Fanuc KAREL source: kt00993.KL

-- PROVISIONAL review KL for V770-1; original PC SHA256 12c16eac051c8f9e1ecef42b03a925e4016cb3948922b7bc4d866e11e08eff63
-- Incomplete behavior may be omitted. Consult companion uncertainty JSON. Do not deploy.
PROGRAM KT00993
%NOLOCKGROUP
VAR
  X : REAL
  Y : REAL
  Z : REAL
  W : REAL
  P : REAL
  R : REAL
-- UNRESOLVED_DECL P1 type=000106
-- UNRESOLVED_DECL P2 type=000106
-- UNRESOLVED_DECL CFG type=00001c
BEGIN
  -- UNRESOLVED_PC offsets 5-20; opcodes 2E,22,32,35
  -- UNRESOLVED_PC offsets 25-40; opcodes 2E,22,32,35
  -- UNRESOLVED_PC offsets 45-60; opcodes 2E,22,32,35
  -- UNRESOLVED_PC offsets 65-80; opcodes 2E,22,32,35
  -- UNRESOLVED_PC offsets 85-145; opcodes 27,27,49,7E,AD,22,22,22,22,22,22,22,76
  -- UNRESOLVED_PC offsets 150-154; opcodes 7F
END KT00993
